# EPICS substitutions: hugo/source/db/empty.substitutions
file "empty.template"
{
  pattern {}
}
